TYPE ST_series :
STRUCT
	data: ARRAY[0..6] OF INT;	
END_STRUCT
END_TYPE

(* stored: Version 1.1.0.1, ProductVersion 3.1.4022.18
   DUT ST_series: Id {1a0b1c5a-580c-4a97-8303-2dd1b2c5b385} *)
